PROGRAM AirVertical_Limit_Switches

VAR
	
	axisAirVertical: AXIS_REF;
    fbAxisPowerAirVertical: MC_Power;
       
	bEnable: BOOL := TRUE;
    fOverride: LREAL := 100;
    		
	biLimFwd_AirVertical AT %I*: BOOL;
	biLimBwd_AirVertical AT %I*: BOOL;

	fbtest:FB_Test;
END_VAR


fbtest(
	axis:=axisAirVertical , 
	fTargetVelocity:=0.3 , 
	fStartPosition:= -4.1, 
	fEndPosition:= 3, 
	nDivisions:= 20 , 
	fbAxisPower:= fbAxisPowerAirVertical );
fbAxisPowerAirVertical(
    Axis:= axisAirVertical,
    Enable:= bEnable,
    Enable_Positive:= biLimFwd_AirVertical, // TRUE, //
    Enable_Negative:= biLimBwd_AirVertical, // TRUE, //
    Override:= fOverride,
    BufferMode:= ,
    Options:= ,
    Status=> ,
    Busy=> ,
    Active=> ,
    Error=> ,
    ErrorID=> );

END_PROGRAM

(* stored: Version 1.1.0.1, ProductVersion 3.1.4024.4
   POU AirVertical_Limit_Switches: Id {97114625-ac17-4a14-8767-b57581610e25}, SpecialFunc None *)
